// TIA Portal V15.1 export
// export: Created 2020-06-12T07:35:41.7880859Z, ExportSetting None, DisplayName Totally Integrated Automation Portal, DisplayVersion V15.1, DisplayName TIA Portal Openness, DisplayVersion V15.1, DisplayName STEP 7 Professional, DisplayVersion V15.1, DisplayName STEP 7 Safety, DisplayVersion V15.1, DisplayName WinCC Advanced, DisplayVersion V15.1
FUNCTION "TimeSrvcs" : Void   // FC39, FBD
TITLE = Time, timesync with HMI and OPs, new time periode
{ S7_Optimized_Access := 'TRUE' }
AUTHOR : atec
FAMILY : COMMON
NAME : TimeSrvc
VERSION : 1.0
// Uhrzeit, Uhrzeitsyncs mit Vis u. OPs, neuer Zeitabschnitt
// stored: SetENOAutomatically False
   VAR_TEMP
      tRetVal : Int;   // Return Value from Siemens Functionblock
      tINT : Int;
   END_VAR
BEGIN

REGION Network 1: Cycle time of previous scan (milliseconds)
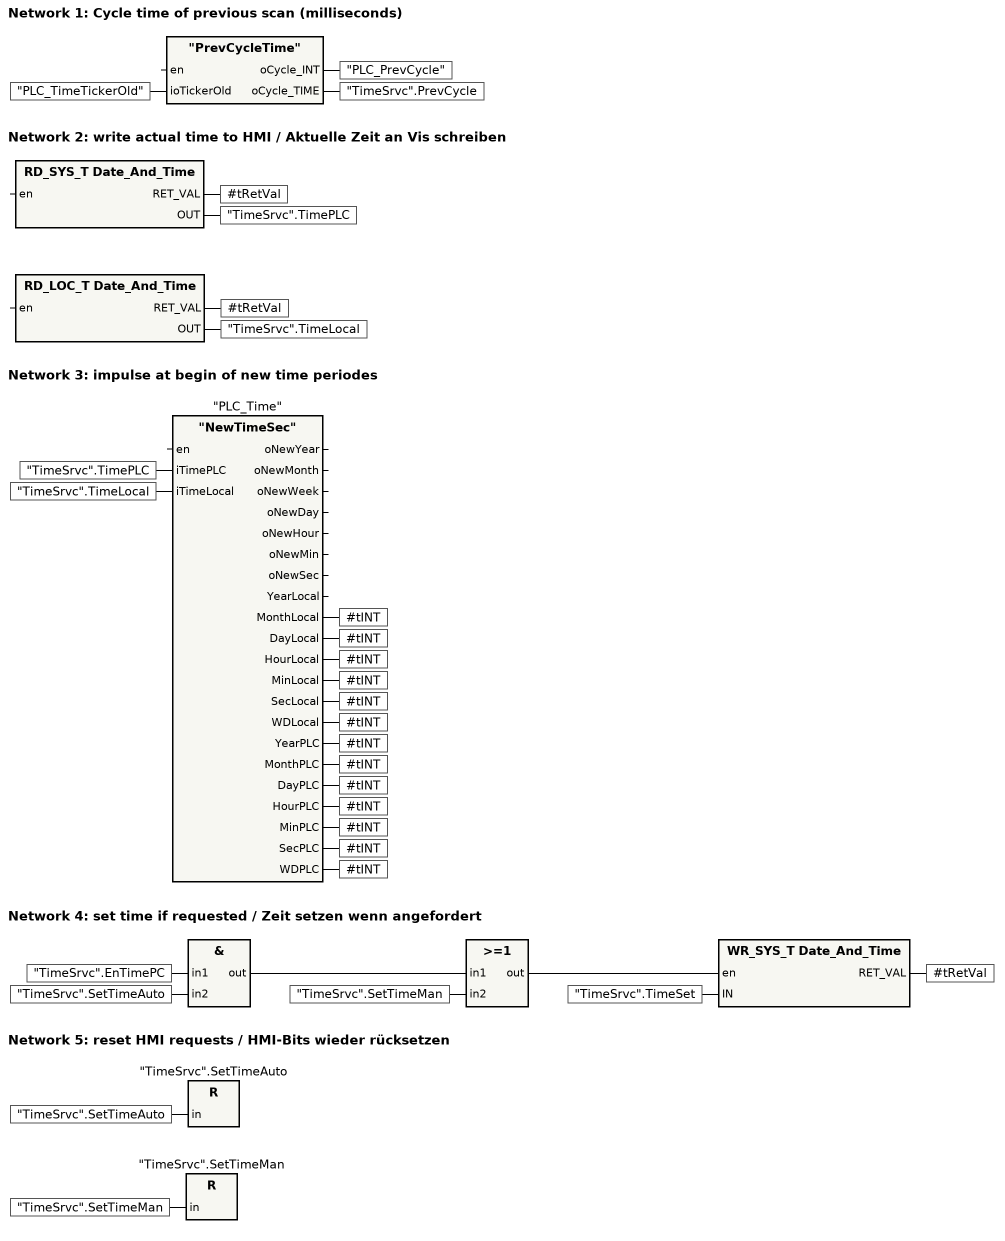
   "PrevCycleTime"(ioTickerOld := "PLC_TimeTickerOld",
                   oCycle_INT => "PLC_PrevCycle",
                   oCycle_TIME => "TimeSrvc".PrevCycle);
END_REGION

REGION Network 2: write actual time to HMI / Aktuelle Zeit an Vis schreiben
   #tRetVal := RD_SYS_T(OUT => "TimeSrvc".TimePLC);
   #tRetVal := RD_LOC_T(OUT => "TimeSrvc".TimeLocal);
END_REGION

REGION Network 3: impulse at begin of new time periodes
   // NOT USED
   "PLC_Time"(iTimePLC := "TimeSrvc".TimePLC,   // "NewTimeSec"
              iTimeLocal := "TimeSrvc".TimeLocal,
              MonthLocal => #tINT,
              DayLocal => #tINT,
              HourLocal => #tINT,
              MinLocal => #tINT,
              SecLocal => #tINT,
              WDLocal => #tINT,
              YearPLC => #tINT,
              MonthPLC => #tINT,
              DayPLC => #tINT,
              HourPLC => #tINT,
              MinPLC => #tINT,
              SecPLC => #tINT,
              WDPLC => #tINT);
END_REGION

REGION Network 4: set time if requested / Zeit setzen wenn angefordert
   IF ("TimeSrvc".EnTimePC AND "TimeSrvc".SetTimeAuto) OR "TimeSrvc".SetTimeMan THEN
       #tRetVal := WR_SYS_T(IN := "TimeSrvc".TimeSet);
   END_IF;
END_REGION

REGION Network 5: reset HMI requests / HMI-Bits wieder rücksetzen
   IF "TimeSrvc".SetTimeAuto THEN "TimeSrvc".SetTimeAuto := FALSE; END_IF;
   IF "TimeSrvc".SetTimeMan THEN "TimeSrvc".SetTimeMan := FALSE; END_IF;
END_REGION
END_FUNCTION
